// TIA Portal project "Niveauregelung" (V15)

(* hardware
DEVICE "S7-1200-Station_1"  S7-1200 Station
   slot 0: "Baugruppenträger_0"  S7-1200 Rack  Rack  V1.0
   slot 1: "PLC_1"  CPU 1214C DC/DC/Rly  6ES7 214-1HG40-0XB0  V4.2
DEVICE "HMI_1"  KTP700 Basic PN
   slot 0: "HMI_1"  KTP700 Basic PN  6AV2 123-2GB03-0AX0  15.0.0.0
   slot 1: "HMI_RT_1"  KTP700 Basic PN  6AV2 123-2GB03-0AX0  15.0.0.0
   slot 5: "HMI_1.IE_CP_1"  PROFINET Interface  15.0.0.0
      slot 1: "PROFINET Schnittstelle_1"  PROFINET Interface
         slot 1: "Port_1"  Port
*)

// ===== PLC "PLC_1"  CPU 1214C DC/DC/Rly =====

VAR_GLOBAL   // PLC tag table "Standard-Variablentabelle"
   "S1" AT %I0.0 : Bool;   // Anlage Start (Schließer)
   "S2" AT %I0.1 : Bool;   // Anlage Stop(Öffner)
   "S3" AT %I0.2 : Bool;   // Störung Quittierung(Schleißer)
   "B1" AT %I0.3 : Bool;   // Füllstand min.(Schließer)
   "B2" AT %I0.4 : Bool;   // Füllstand mitte(Schließer)
   "B3" AT %I0.5 : Bool;   // Füllstand max.(Öffner)
   "F1" AT %I0.6 : Bool;   // Motorschutz Motor 1(Öffner)
   "F2" AT %I0.7 : Bool;   // Motorschutz Motor 2(Öffner)
   "Q1" AT %Q0.0 : Bool;   // Motor M1
   "Q2" AT %Q0.1 : Bool;   // Motor M2
   "P1" AT %Q0.2 : Bool;   // Anlage Störung
   "P2" AT %Q0.3 : Bool;   // Anlage Ein
   "P3" AT %Q0.4 : Bool;   // Füllstand min.
   "Merker Füllstand max." AT %M0.0 : Bool;
   "Merker Füllstand mitte" AT %M0.1 : Bool;
   "Merker Füllstand min" AT %M0.2 : Bool;
   "Sammelstörung" AT %M0.3 : Bool;
   "Merker 1 Störung" AT %M0.4 : Bool;
   "Merker P1" AT %M0.5 : Bool;
   "Merker Anlage Betriebsbereit" AT %M0.6 : Bool;
END_VAR

DATA_BLOCK "HMI"   // DB3
{ S7_Optimized_Access := 'TRUE' }
VERSION : 0.1
   VAR
      Start : Bool;
      Stop : Bool;
   END_VAR
BEGIN
END_DATA_BLOCK

// folder: System blocks/Program resources

DATA_BLOCK "IEC_Timer_0_DB"   // DB1
{ S7_Optimized_Access := 'TRUE' }
AUTHOR : Simatic
FAMILY : IEC
NAME : IEC_TMR
VERSION : 1.0
// stored: InstanceOfName IEC_TIMER
"IEC_TIMER"
BEGIN
END_DATA_BLOCK

DATA_BLOCK "IEC_Timer_0_DB_1"   // DB2
{ S7_Optimized_Access := 'TRUE' }
AUTHOR : Simatic
FAMILY : IEC
NAME : IEC_TMR
VERSION : 1.0
// stored: InstanceOfName IEC_TIMER
"IEC_TIMER"
BEGIN
END_DATA_BLOCK

DATA_BLOCK "IEC_Timer_0_DB_2"   // DB4
{ S7_Optimized_Access := 'TRUE' }
AUTHOR : Simatic
FAMILY : IEC
NAME : IEC_TMR
VERSION : 1.0
// stored: InstanceOfName IEC_TIMER
"IEC_TIMER"
BEGIN
END_DATA_BLOCK

DATA_BLOCK "IEC_Timer_0_DB_3"   // DB5
{ S7_Optimized_Access := 'TRUE' }
AUTHOR : Simatic
FAMILY : IEC
NAME : IEC_TMR
VERSION : 1.0
// stored: InstanceOfName IEC_TIMER
"IEC_TIMER"
BEGIN
END_DATA_BLOCK

DATA_BLOCK "IEC_Timer_0_DB_4"   // DB6
{ S7_Optimized_Access := 'TRUE' }
AUTHOR : Simatic
FAMILY : IEC
NAME : IEC_TMR
VERSION : 1.0
// stored: InstanceOfName IEC_TIMER
"IEC_TIMER"
BEGIN
END_DATA_BLOCK

// folder: (top level)

FUNCTION "Niveauregelung" : Void   // FC1, FBD
TITLE = Niveauregelung
{ S7_Optimized_Access := 'TRUE' }
VERSION : 0.1
BEGIN

REGION Network 1: Anlage Betriebsbereit
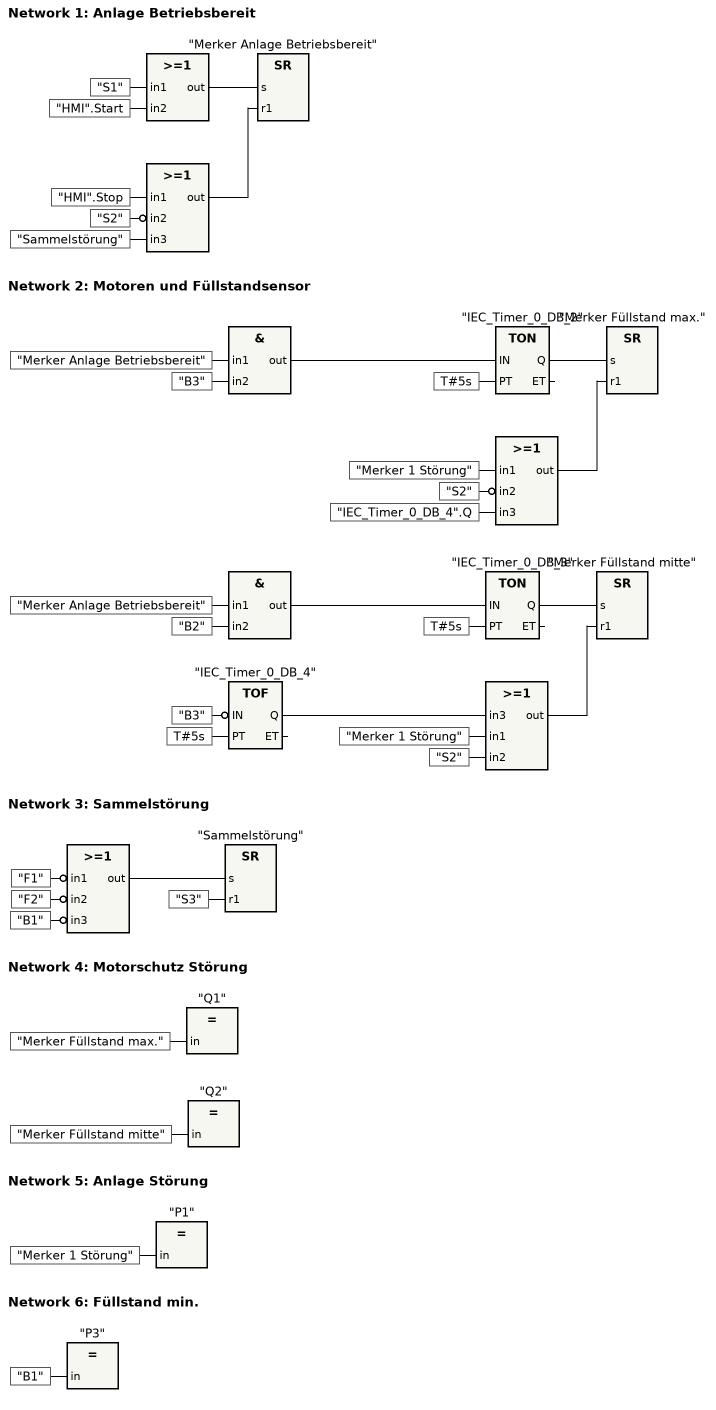
   IF "S1" OR "HMI".Start THEN
       "Merker Anlage Betriebsbereit" := TRUE;   // SR flip-flop
   END_IF;
   IF "HMI".Stop OR NOT "S2" OR "Sammelstörung" THEN "Merker Anlage Betriebsbereit" := FALSE; END_IF;
END_REGION

REGION Network 2: Motoren und Füllstandsensor
   "IEC_Timer_0_DB_2".TON(IN := "Merker Anlage Betriebsbereit" AND "B3", PT := T#5s);
   IF "IEC_Timer_0_DB_2".Q THEN
       "Merker Füllstand max." := TRUE;   // SR flip-flop
   END_IF;
   IF "Merker 1 Störung" OR NOT "S2" OR "IEC_Timer_0_DB_4".Q THEN "Merker Füllstand max." := FALSE; END_IF;
   "IEC_Timer_0_DB_3".TON(IN := "Merker Anlage Betriebsbereit" AND "B2", PT := T#5s);
   "IEC_Timer_0_DB_4".TOF(IN := NOT "B3", PT := T#5s);
   IF "IEC_Timer_0_DB_3".Q THEN
       "Merker Füllstand mitte" := TRUE;   // SR flip-flop
   END_IF;
   IF "IEC_Timer_0_DB_4".Q OR "Merker 1 Störung" OR "S2" THEN "Merker Füllstand mitte" := FALSE; END_IF;
END_REGION

REGION Network 3: Sammelstörung
   IF NOT "F1" OR NOT "F2" OR NOT "B1" THEN
       "Sammelstörung" := TRUE;   // SR flip-flop
   END_IF;
   IF "S3" THEN "Sammelstörung" := FALSE; END_IF;
END_REGION

REGION Network 4: Motorschutz Störung
   "Q1" := "Merker Füllstand max.";
   "Q2" := "Merker Füllstand mitte";
END_REGION

REGION Network 5: Anlage Störung
   "P1" := "Merker 1 Störung";
END_REGION

REGION Network 6: Füllstand min.
   "P3" := "B1";
END_REGION
END_FUNCTION

ORGANIZATION_BLOCK "Main"   // OB1, LAD, ProgramCycle
TITLE = "Main Program Sweep (Cycle)"
{ S7_Optimized_Access := 'TRUE' }
VERSION : 0.1
   VAR_INPUT
      Initial_Call : Bool;   // Initial call of this OB
      Remanence : Bool;   // =True, if remanent data are available
   END_VAR
BEGIN

REGION Network 1
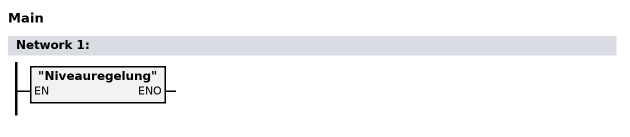
   RUNG wire#powerrail
      "Niveauregelung"()
   END_RUNG
   // the same network as SCL:
   "Niveauregelung"();
END_REGION
END_ORGANIZATION_BLOCK

(* ===== HMI "HMI_RT_1" =====
system functions are stored by id; their names below are inferred from use
connection "HMI_Verbindung_1": ETHERNET, SMART_S7_1200_OMS

HMI tags "Standard-Variablentabelle"
   "B3" : Bool = PLC B3 AT %I0.5, 100 ms
   "B1" : Bool = PLC B1 AT %I0.3, 100 ms
   "B2" : Bool = PLC B2 AT %I0.4, 100 ms
   "Start" : Bool = PLC HMI.Start, 1 s
   "Stop" : Bool = PLC HMI.Stop, 1 s

screen "Bild_1" 800x480
   Button "Schaltfläche_1" at 55,147 size 200x84; TextOff 'Start'
      on Press: function_b14e0dd5("Start", 0)
   Button "Schaltfläche_2" at 55,284 size 200x84; TextOff 'Stop'
      on Press: function_b14e0dd5("Stop", 0)
   Circle "Kreis_2" at 627,120 size 50x50
      Appearance <- "B3"
   Circle "Kreis_3" at 627,274 size 50x50
      Appearance <- "B2"
   Circle "Kreis_4" at 596,375 size 50x50
      Appearance <- "B1"
   TextField "Textfeld_1" at 55,14 size 133x23; Text 'Niveauregelung'
   TextField "Textfeld_3" at 59,46 size 309x23; Text 'Prüflingsnummer 007, am 21.06.2020'
   TextField "Textfeld_2" at 655,386 size 26x23; Text 'B1'
   TextField "Textfeld_4" at 686,284 size 26x23; Text 'B2'
   TextField "Textfeld_5" at 686,134 size 26x23; Text 'B3'
   GraphicView "Grafikanzeige_1" at 398,69 size 198x379; Picture "Grafik_1"
*)